FUNCTION_BLOCK INTERNAL FB_DisconnectedState IMPLEMENTS I_State
VAR
	pMachine		: POINTER TO FB_Machine; // Points to the state machine (THIS)
	fVSensors		: ARRAY[0..1] OF REAL; 
END_VAR

METHOD PUBLIC Check
VAR
	fInputVoltage 		: REAL; 
END_VAR
THIS^.ResetContactors(); //THE CONTACTORS NEED TO ALWAYS BE OPEN IN THIS STATE
fVSensors := THIS^.pMachine^.VSensors;
fInputVoltage := fVSensors[0];

IF (fInputVoltage >= THIS^.pMachine^.MinV) THEN
	THIS^.pMachine^.Message := '[DISCONNECTED] The input voltage is >= than the minimum voltage. $0A WAITING FOR ACKNOWLEDGEMENT TO ENTER IDLE STATE;';
ELSE 
	THIS^.pMachine^.Message := '[DISCONNECTED]The input voltage is <= than the minimum voltage.';
END_IF
END_METHOD

PROPERTY PUBLIC Description : STRING
GET
Description := 'DISCONNECTED';
END_GET
END_PROPERTY

METHOD PUBLIC FB_init
VAR_INPUT
	bInitRetains 	: BOOL; // if TRUE, the retain variables are initialized (warm start / cold start)
	bInCopyCode 	: BOOL;  // if TRUE, the instance afterwards gets moved into the copy code (online change)
	pMachine		: POINTER TO FB_Machine; // Points to the state machine (THIS)
END_VAR
THIS^.pMachine := pMachine;
END_METHOD

METHOD PUBLIC PressButton 
VAR
	//fbIdleSTate		: FB_IdleState(THIS^.pMachine); => variable for changing state method that causes a PLC bug
	fInputVoltage		: REAL; 
END_VAR
fVSensors := THIS^.pMachine^.VSensors;
fInputVoltage := fVSensors[0];

IF (fInputVoltage >= THIS^.pMachine^.MinV) THEN
		//THIS^.pMachine^.SetState(fbIdleState); => changing state method that causes a PLC bug
		THIS^.pMachine^.Message := '[DISCONNECTED] Acknowledge button has been pressed. $0A SYSTEM ENTERS IDLE STATE.';
		THIS^.pMachine^.SetState(THIS^.pMachine^.IdleState);
END_IF
END_METHOD

METHOD PUBLIC PressDischarge
END_METHOD

METHOD PUBLIC Reset
END_METHOD

METHOD PUBLIC ResetContactors
VAR
	nIdx					: INT := 0; 
	bBypassContactors		: ARRAY[0..1] OF BOOL; 
	bMainContactors			: ARRAY[0..1] OF BOOL; 
END_VAR
FOR nIdx := 0 TO 1 BY 1 DO 
	bBypassContactors[nIdx] := FALSE;
	bMainContactors[nIdx] := FALSE; 
END_FOR

THIS^.pMachine^.BypassContactors := bBypassContactors; // Reset every contactor 
THIS^.pMachine^.MainContactors := bMainContactors;
END_METHOD

METHOD PUBLIC Stop
THIS^.pMachine^.SetState(THIS^.pMachine^.ErrorState);
END_METHOD

METHOD PUBLIC TimerDone
END_METHOD

END_FUNCTION_BLOCK

(* stored: Version 1.1.0.1, ProductVersion 3.1.4024.12
   POU FB_DisconnectedState: Id {b6c9100b-ee0f-440e-b30d-6ce4ff78067b}, SpecialFunc None
   Method Check: Id {f7b4c791-cd0a-45fe-88c9-0fe129bd6102}
   Property Description: Id {3242d7fd-7be6-46ed-8cdb-6f18a3c23c7f}
   Get Get: Id {59bb9789-25c7-40b4-913d-675faf0da855}
   Method FB_init: Id {740eb518-5aff-468b-8d2a-587ff6255015}
   Method PressButton: Id {e6c89707-d232-4033-95e2-33255f005dce}
   Method PressDischarge: Id {13d2dd19-2000-4709-9874-14f10538b54a}
   Method Reset: Id {5527b193-c28b-4d9e-b368-bee68cae1ff1}
   Method ResetContactors: Id {57b6047e-2a92-40e6-b4a9-31e4fbc5e8b0}
   Method Stop: Id {4ec2f479-c802-41f1-985e-64350926edc5}
   Method TimerDone: Id {8beb5e78-39a9-4f59-8783-fd5f819a3f39} *)
